TYPE T_SIM_LAMP_STAT :
STRUCT
	bInitialised:	BOOL	:= FALSE;						(* If TRUE, lamp simulator is initialised *)

	nErrorCode: 	E_LAMP_ERROR 	:= E_LAMP_ERROR.SIM_NOT_INITIALISED;	(* Error code *)
	sErrorText: 	STRING 	:= 'NOT INITIALISED'; 			(* Error text *)
	sStatus: 		STRING 	:= 'ERROR'; 					(* Lamp status in textual form, e.g. 'OFF' *)
END_STRUCT
END_TYPE

(* stored: Version 1.1.0.1, ProductVersion 3.1.4022.16
   DUT T_SIM_LAMP_STAT: Id {91af19d4-208f-48f7-a423-e4ef68fbafcd} *)
